FUNCTION_BLOCK HB_M2S
VAR_INPUT
	Dur : TIME;
END_VAR
VAR_OUTPUT
	OK : BOOL;
	ET : TIME;
END_VAR
VAR
	Timer : TON;
	Count_Last : INT;
END_VAR
VAR_IN_OUT
	Counter : USINT;
END_VAR
VAR // added by the converter: edge detectors and wires of the graphical bodies
    _w1, _w2 : BOOL;
END_VAR

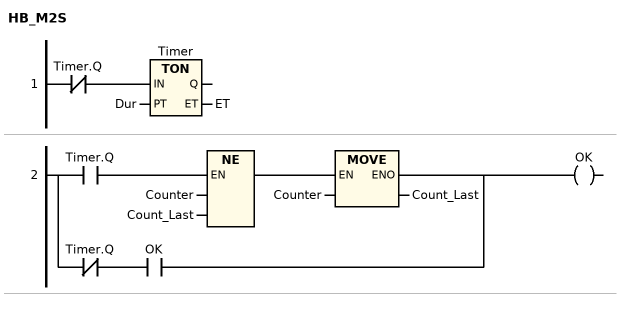
// NETWORK 1
Timer(IN := NOT Timer.Q, PT := Dur, ET => ET); // TON

// NETWORK 2
_w1 := NOT Timer.Q AND OK;
IF NOT _w1 THEN
    _w2 := Timer.Q AND Counter <> Count_Last;
    IF _w2 THEN Count_Last := Counter; END_IF
    _w1 := _w2;
END_IF
OK := _w1;

END_FUNCTION_BLOCK

(* stored: Version 1.1.0.1, ProductVersion 3.1.4024.9
   POU HB_M2S: Id {6b5c44ae-b2bf-4578-b20e-e4342a01bd4e}, SpecialFunc None *)
